Fanuc KAREL source: f_defgrp_t.kl

PROGRAM F_DEFGRP_T
%DEFGROUP = 2
%CRTDEVICE
%DELAY = 20
VAR
  p : XYZWPR IN GROUP[2]
  i : INTEGER
BEGIN
  $SPEED = 100
  MOVE TO p
  WITH $SPEED = 200 MOVE TO p
  WRITE('x', i, CR)
  READ(i)
END F_DEFGRP_T
